(* IEC 61131-3 sources: programs/VI-54/VI-54_20171205/VI-54_20171205/Stations/PLC_VI54/VI-54_171014/Class/PauseClass, 1 file *)

(* ---- PauseClass.st ---- *)
(*!
<Class
	Name               = "PauseClass"
	Revision           = "0.0"
	RealtimeTask       = "false"
	CyclicTask         = "false"
	BackgroundTask     = "true"
	Sigmatek           = "false"
	OSInterface        = "false"
	HighPriority       = "false"
	Automatic          = "false"
	UpdateMode         = "Prescan"
	SharedCommandTable = "true"
	Objectsize         = "(780,480)">
	<Channels>
		<Server Name="Comm" Visualized="false" Initialize="false" WriteProtected="true" Retentive="false"/>
		<Server Name="In_ExternPauseDelay" Visualized="true" Initialize="true" WriteProtected="false" Retentive="File"/>
		<Server Name="In_ExternPauseOptions" Visualized="true" Initialize="true" WriteProtected="false" Retentive="File"/>
		<Server Name="In_InternPauseDelay" Visualized="true" Initialize="true" WriteProtected="false" Retentive="File"/>
		<Server Name="In_InternPauseOptions" Visualized="true" Initialize="true" WriteProtected="false" Retentive="File"/>
		<Server Name="Out_PauseDelay" Visualized="true" Initialize="true" WriteProtected="false" Retentive="File"/>
		<Server Name="Out_PauseOptions" Visualized="true" Initialize="true" WriteProtected="false" Retentive="File"/>
		<Client Name="In_Extern_Pause" Required="false" Internal="false"/>
		<Client Name="In_Intern_Pause" Required="false" Internal="false"/>
		<Client Name="Out_Pause" Required="false" Internal="false"/>
		<Client Name="Standard1" Required="true" Internal="true"/>
	</Channels>
	<Separators>
		<Servers>
			<SepChn Position="1"/>
			<SepChn Position="4"/>
			<SepChn Position="7"/>
		</Servers>
	</Separators>
	<Network Name="PauseClass">
		<!-- List of Components in this network -->
		<Components>
			<Object
				Name           = "Standard1"
				Class          = "Standard"
				Position       = "(150,120)"
				Visualized     = "false"
				BackgroundTime = "1000 ms">
				<Channels>
					<Server Name="ClassSvr"/>
				</Channels>
			</Object>
		</Components>
		<Comments>
		</Comments>
		<!-- List of Connections in this network -->
		<Connections>
			<Connection Source="this.Standard1" Destination="Standard1.ClassSvr"/>
		</Connections>
		<!-- Headerfiles -->
		<Options>
		</Options>
	</Network>
</Class>
*)
PauseClass : CLASS
	TYPE
	  ePauseOptions :  //! <Type Public="true" Name="ePauseOptions"/>
	  (
	    eNormalyClosed,
	    eNormalyOpen,
	    ePuls
	  )$UDINT;
	END_TYPE
  //Servers:
	Comm 	: SvrChCmd_DINT;
	In_InternPauseOptions 	: SvrCh_ePauseOptions_PTofCls_PauseClass;
	In_InternPauseDelay 	: SvrCh_DINT;
	In_ExternPauseOptions 	: SvrCh_ePauseOptions_PTofCls_PauseClass;
	In_ExternPauseDelay 	: SvrCh_DINT;
	Out_PauseOptions 	: SvrCh_ePauseOptions_PTofCls_PauseClass;
	Out_PauseDelay 	: SvrCh_DINT;
  //Clients:
	In_Intern_Pause 	: CltCh_DINT;
	In_Extern_Pause 	: CltCh_DINT;
	Out_Pause 	: CltCh_DINT;
	Standard1 	: CltChCmd_Standard;
  //Variables:
		ExternPause 	: DINT;
		InternPause 	: DINT;
  //Functions:

	FUNCTION VIRTUAL GLOBAL Background
		VAR_INPUT
			EAX 	: UDINT;
		END_VAR
		VAR_OUTPUT
			state (EAX) 	: UDINT;
		END_VAR;

	FUNCTION GLOBAL PauseInternal
		VAR_INPUT
			PauseState 	: ePauseOptions;
			iPauseSignal 	: DINT;
		END_VAR;

	FUNCTION GLOBAL PauseExternal
		VAR_INPUT
			PauseState 	: ePauseOptions;
			iPauseSignal 	: DINT;
		END_VAR;

	FUNCTION GLOBAL GetPauseState
		VAR_OUTPUT
			State 	: DINT;
		END_VAR;
  //Tables:
	FUNCTION @STD
		VAR_OUTPUT
			ret_code	: CONFSTATES;
		END_VAR;
	FUNCTION GLOBAL TAB @CT_;
END_CLASS;

#pragma using Standard

FUNCTION VIRTUAL GLOBAL PauseClass::Background
	VAR_INPUT
		EAX 	: UDINT;
	END_VAR
	VAR_OUTPUT
		state (EAX) 	: UDINT;
	END_VAR

  // Read input
  // if IsClientConnected(#In_Intern_Pause) then
    In_Intern_Pause := In_Intern_Pause.Read();
    In_Extern_Pause := In_Extern_Pause.Read();
  // else
  //  In_Intern_Pause := 1;
  //end_if;

  // Write output
  if IsClientConnected(#Out_Pause) then
    Out_Pause.Write(input:= Out_Pause);
  end_if;

  // Open methodes
  PauseInternal(PauseState:= In_InternPauseOptions, iPauseSignal:= In_Intern_Pause);
  PauseExternal(PauseState:= In_ExternPauseOptions, iPauseSignal:= In_Extern_Pause);

	state := READY;

END_FUNCTION

FUNCTION GLOBAL PauseClass::PauseInternal
	VAR_INPUT
		PauseState 	: ePauseOptions;
		iPauseSignal 	: DINT;
	END_VAR

  case PauseState of
    eNormalyClosed:
      InternPause := (iPauseSignal = 1);
    eNormalyOpen:
      InternPause := (iPauseSignal = 0);
    ePuls:
      if Standard1.R_TRIG(CLK:= iPauseSignal) then
        InternPause := (InternPause xor 1);
      end_if;
  end_case;

END_FUNCTION

FUNCTION GLOBAL PauseClass::PauseExternal
	VAR_INPUT
		PauseState 	: ePauseOptions;
		iPauseSignal 	: DINT;
	END_VAR

  case PauseState of
    eNormalyClosed:
      ExternPause := (iPauseSignal = 1);
    eNormalyOpen:
      ExternPause := (iPauseSignal = 0);
    ePuls:
      if Standard1.R_TRIG(CLK:= iPauseSignal) then
        ExternPause := (ExternPause xor 1);
      end_if;
  end_case;

END_FUNCTION

FUNCTION GLOBAL PauseClass::GetPauseState
	VAR_OUTPUT
		State 	: DINT;
	END_VAR

  State := (InternPause = 1 | ExternPause = 1);

END_FUNCTION
